PROGRAM P_Outputs
VAR
	stValveOutput : FB_ValveOutput;
END_VAR

stValveOutput(
	bEnable := (G_Work.eStatus = E_Status.Running),
	stParam := G_Parameters.stParam,
	fNormalizedInput := G_VirtualControlBox.fJoystickY,
	bEnableValveOutput => G_Outputs.stValveOutput.bEnable,
	nOutput => G_Outputs.stValveOutput.nValveOutput
);

END_PROGRAM

(* stored: Version 1.1.0.1, ProductVersion 3.1.4024.10
   POU P_Outputs: Id {340d1cdc-77aa-4d41-803b-eca0e7407e8a}, SpecialFunc None *)
